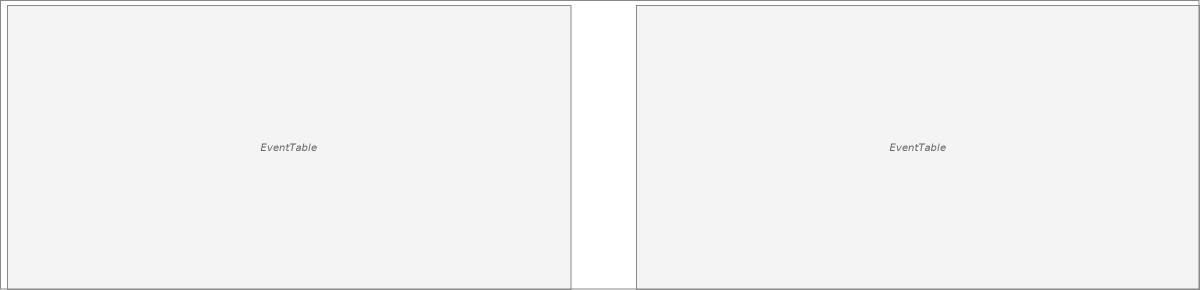
VISUALIZATION Visualization  // 1200x290
    EventTable (636,5 564x285)
        p1690906150: Class
        p3258520714: Date
        p2231227367: Time
        p3993844394: Message
        p2076579579: Details
        p3558512729: MAIN.LoggedEvents
        p3921149237: m_pDataArray..pArray
    EventTable (7,5 564x285)
        p1690906150: Class
        p3258520714: Date
        p2231227367: Time
        p3993844394: Message
        p2076579579: Details
        p3558512729: MAIN.fbReadTc3Events.aEvents
        p3921149237: m_pDataArray..pArray
END_VISUALIZATION

(* stored: Version 1.1.0.1
   Visu Visualization: Id {2fbb7686-a988-4f89-a599-93a43e34461e} *)
